Universal Robots PolyScope program: translation_sample_servoj_egg.urp

Program translation_sample_servoj_egg (installation=servoj2 directory=/programs/servoj createdIn=3.2.19275 lastSavedIn=5.13.1 robotSerialNumber=20195380017)
Calibrated DH parameters: a=[-0.000005, -0.241897, -0.163857, -0.000004, -0.000042, 0]; d=[0.15198, 4.092034, -18.51686, 14.555458, 0.085328, 0.092191]; alpha=[1.570113, -0.007378, -0.009451, 1.571508, -1.571142, 0]; deltaTheta=[-0.000001, -0.124164, 0.818102, -0.693964, 0.000084, 0]
InitVariablesNode
BeforeStart
  MoveJ speed 50 deg/s, acceleration 40 deg/s^2 (useActiveTCP=true) feature=Base
    Waypoint 路点_1: TCP in base x=19.811 y=-362.643 z=97.756 mm, rx=3.1282 ry=-0.0129 rz=-0.074 rad; joints [-62.12, -93.328, -80.246, -97.094, 86.866, -150.782] deg; TCP offset x=1.059 y=22.521 z=227.924 mm, rx=0 ry=0 rz=0 rad
  joints := get_actual_joint_positions()
  home := get_actual_tcp_pose()
  Script: write_output_boolean_register(0, False )
  SuppressedNode
    Script: write_input_interger_register(0,0)
  Wait Sleep waitTime=0.01
  Script: popup("Registers reset, run PC code and then click Continue",title="Hi Daniel",blocking= True )
  mode := 0
Robot Program (runOnlyOnce=false)
  Script: write_output_boolean_register(0, True )
  Script: sync()
  Loop While (checkContinuously=false) expression=mode<3
    Loop While (checkContinuously=false) expression=mode≟1
      MoveJ speed 60 deg/s, acceleration 80 deg/s^2 (useActiveTCP=true) feature=Base
        Waypoint Variable (Variable): variable(name=joints)
      Script: write_output_boolean_register(0, False )
      Script: sync()
    Loop While (checkContinuously=false) expression=mode≟2
      Script: servoj(joints, 0, 0, 0.03, 0.9, 1800)
    Loop While (checkContinuously=false) expression=mode≟3
      Halt
  Script: sync()
Thread Thread_1 (runOnlyOnce=false)
  tmp := p[0,0,0,0,0,0]
  tmp := p[0,0,0,0,0,0]
  maxX := 0.18
  maxY := 0.18
  maxZ := 0.06
  Loop Forever
    Script file /programs/pose_register.script
      | tmp[0]=read_input_float_register(0)
      | tmp[1]=read_input_float_register(1)
      | tmp[2]=read_input_float_register(2)
      | tmp[3]=read_input_float_register(3)
      | tmp[4]=read_input_float_register(4)
      | tmp[5]=read_input_float_register(5)
    SuppressedNode
      If mode≟2
        tmp := pose_trans(home, tmp)
        SuppressedNode
          Script: tmp=pose_trans(get_actual_tcp_pose(), tmp)
    SuppressedNode
      tmp := pose_trans(home, tmp)
    SuppressedNode
      tmp := pose_trans(get_actual_tcp_pose(), tmp)
    SuppressedNode
      diff := pose_trans(pose_inv(平面_3), tmp)
    SuppressedNode
      Popup Message (haltProgram=true message=1 inputType=Text)
    SuppressedNode
      If diff[0]≤0
        Script: diff[0] =0
    SuppressedNode
      If diff[1]≤0
        Script: diff[1] =0
    SuppressedNode
      If diff[2]≤0
        Script: diff[2] =0
    SuppressedNode
      If diff[0]   ≥  maxX
        Script: diff[0] =maxX
    SuppressedNode
      If diff[1] ≥ maxY
        Script: diff[1]=maxY
    SuppressedNode
      If diff[2]≥maxZ
        Script: diff[2]=maxZ
    SuppressedNode
      temp := pose_trans(平面_3, diff)
    joints := get_inverse_kin(p[tmp[0],tmp[1],tmp[2],tmp[3],tmp[4],tmp[5]],get_actual_joint_positions())
    Script: sync()
    mode := read_input_integer_register(0)
    Script: sync()
